Fanuc KAREL source: kt00257.KL

-- PROVISIONAL review KL for V1013-1; original PC SHA256 842b5d39eea4e3cea3adc34c395773c7dd6103d2c7dbc7dfc48556137e3e956f
-- Incomplete behavior may be omitted. Consult companion uncertainty JSON. Do not deploy.
PROGRAM KT00257
%NOLOCKGROUP
VAR
  I1 : INTEGER
  I2 : INTEGER
  OUT : BOOLEAN
BEGIN
  -- UNRESOLVED_PC offsets 5-16; opcodes 2E,23
  -- UNRESOLVED_PC offsets 21-32; opcodes 2E,23
  -- UNRESOLVED_PC offsets 37-48; opcodes 2E,23
  -- UNRESOLVED_PC offsets 53-64; opcodes 2E,23
  -- UNRESOLVED_PC offsets 69-88; opcodes 21,21,57,23
  -- UNRESOLVED_PC offsets 93-97; opcodes 7F
END KT00257
